TYPE ST_systemState :
STRUCT
	bAnlageEin: BOOL;
	bAnlageAus: BOOL;
END_STRUCT
END_TYPE

(* stored: Version 1.1.0.1
   DUT ST_systemState: Id {e8bfe8bd-2321-4c88-9dda-b8aa9cbab3b3} *)
